//==================================================================================================
//							Beckhoff Automation Poland
//									21.05.2018
//	Struktura zawierajaca I/O odpowiedniego bloku
//  v1.0	|| TC v 3.1.4022.16		|| - pierwsza wersja
//==================================================================================================
TYPE ST_FBMotorMonitoringIO:
STRUCT
	bReset							: BOOL;								// Reset FB
	rTorqueLimit					: REAL		:=	500; 				// Bipolar torque limit: 0-500%, resolution 0.1%, value goes to: 16#6072 (Ch A)/ 16#6872 (Ch B)

	bError							: BOOL; 							// General error: parameter or CoE read.
																		// If bError = TRUE and bInitialized = FALSE - error during read motor data.
																		// If bError = TRUE and bInitialized = TRUE and (iAdsErrId <> 0 or iCANopenErrId <> 0) then I2T read error
																		// If bError = TRUE and bInitialized = TRUE and iAdsErrId = 0 and iCANopenErrId = 0 then parameter error: rTorqueLimit outside permitted range rTorqueLimitLow..rTorqueLimitHigh or Empty stDriveRef
	uiAdsErrId						: UINT;								// Forwarded output FB_CoERead_ByDriveRef
	uiSecErrId						: UINT;								// Sercos Error ID for AX5000, CanOpen error ID for AX8000
	bInitialized					: BOOL;								// TRUE - Motor data read without errors, so it's possible to calculate torqe and current values in metric units
	bWarning						: BOOL;								// rCurrentF > rWarningCurrent, be aware to be over permitted range
	rWarningCurrent					: REAL; 							// Continuous Stall Current - motor parameter: 16#6075 (Ch A)/ 16#6875 (Ch B); scalled: [A]
	rTorquePerc						: REAL;								// [%]
	rTorquePercMax					: REAL;								// Max [%]
	rTorque							: REAL; 							// [Nm]
	rTorqueF						: REAL;								// Filtered [Nm]
	rTorqueMax						: REAL;								// Max [Nm]
	rCurrent						: REAL; 							// [A]
	rCurrentF						: REAL;								// Filtered [A]
	rCurrentMax						: REAL;								// Max [A]
	rI2T							: REAL; 							// Thermal Motor Utilization: 16#32C1:02 (Ch A)/ 16#36C1:02 (Ch B); units: [%]
	rI2TMax							: REAL; 							// Max % Nominal
END_STRUCT
END_TYPE

(* stored: Version 1.1.0.1, ProductVersion 3.1.4026.13, FileIdentifier c4d4278318e81165b4bfc8221957a670923cc747, FileSignature 2aead112a4af61a8873d50925886d8ae69dd0b1fde8455716bfd415031107f8edb1bd69a48d9a6c3e9ab9e37f2bb9ff4bb07ea52f717fe7e5c7cc8050d8980fed379a9854d3f83c1343ec3ee414fe51ff6338cb54693a3d93e9e6663df8727dc288fbbd219a318f61c6bad4bf78e9b3fdac4dfc474cf6d8ac7b2f3c4cb841eee9ab90e6a930a788bdabe9b5e0bb7ebc6d891902603cc88af65e12284a4b5dad15356365e796ce8ab91913767e55fed657ac3d44a9b6a9571ea0d9722baceb1fce05b5ac9debb801fd0a18888f4ed1baf5564ddbae6dc37b1c4625a2a21b4626b51bff6fd017247a6503252cff359f8e00a3336cfc1d0d6179231245703975ee0
   DUT ST_FBMotorMonitoringIO: Id {fd46209f-d900-476c-a1cf-055b86bee058} *)
